FUNCTION_BLOCK FB_StringBuilder
VAR
	_value : T_MaxString;
END_VAR

METHOD Append : REFERENCE TO FB_StringBuilder
VAR_INPUT
	value : T_MaxString;
END_VAR
_value := CONCAT(_value, value);

Append REF= THIS^;
END_METHOD

METHOD Clear : REFERENCE TO FB_StringBuilder
VAR_INPUT
END_VAR
_value := '';

Clear REF= THIS^;
END_METHOD

METHOD GetString : T_MaxString
VAR_INPUT
END_VAR
GetString := _value;
END_METHOD

END_FUNCTION_BLOCK

(* stored: Version 1.1.0.1
   POU FB_StringBuilder: Id {2c840a46-1d54-4419-9eea-7ea5d3d0e2ad}, SpecialFunc None
   Method Append: Id {1de5ab37-aec6-4e47-9b43-ebab6d307315}
   Method Clear: Id {5eeb5268-f490-4507-ac56-f7ad9465c6bf}
   Method GetString: Id {8d3ddc0a-f501-495c-b92b-84688db116ba} *)
